(* IEC 61131-3 sources: RL_MAR/experiments/comparison/autoplc/results/gpt-4o-mini_20260511_164212/med_83, 1 file *)

(* ---- med_83_1.st ---- *)
FUNCTION_BLOCK AmusementRideControl
    VAR_INPUT
        StartButton : BOOL; (* Start button input *)
        StopButton : BOOL; (* Emergency stop button input *)
        SpeedSensor : REAL; (* Speed sensor input (RPM) *)
        SafetySensor : BOOL; (* Safety sensor status *)
    END_VAR

    VAR_OUTPUT
        MotorOn : BOOL := FALSE; (* Motor control output *)
        BrakeOn : BOOL := TRUE; (* Brake control output *)
    END_VAR

    VAR
        SpeedLimit : REAL := 60.0; (* Maximum allowed speed in RPM *)
    END_VAR

    // Initialization
    IF StopButton THEN
        // Emergency Stop State
        MotorOn := FALSE;
        BrakeOn := TRUE;
    ELSE
        // Check Start Conditions
        IF StartButton AND NOT StopButton AND (SpeedSensor <= SpeedLimit) AND SafetySensor THEN
            MotorOn := TRUE;
            BrakeOn := FALSE;
        ELSE
            MotorOn := FALSE;
            BrakeOn := TRUE;
        END_IF;

        // Monitor Normal Operation
        IF MotorOn THEN
            IF (SpeedSensor > SpeedLimit) OR NOT SafetySensor THEN
                MotorOn := FALSE;
                BrakeOn := TRUE;
            END_IF;
        END_IF;
    END_IF;

    // Default State (Fail-Safe)
    IF NOT StartButton AND NOT StopButton THEN
        BrakeOn := TRUE;
        MotorOn := FALSE;
    END_IF;

END_FUNCTION_BLOCK
